(* CoDeSys 2.3 project: seven segment P1.pro *)
(* Libraries: STANDARD.LIB 25.11.03 12:18:06, IECSFC.LIB 25.11.03 12:18:06, ANALYZATION.LIB 25.11.03 12:18:06 *)

(* POU PLC_PRG, LD *)
PROGRAM PLC_PRG
VAR
	ix0: BOOL;
	a: WORD;
	count: CTUD;
END_VAR
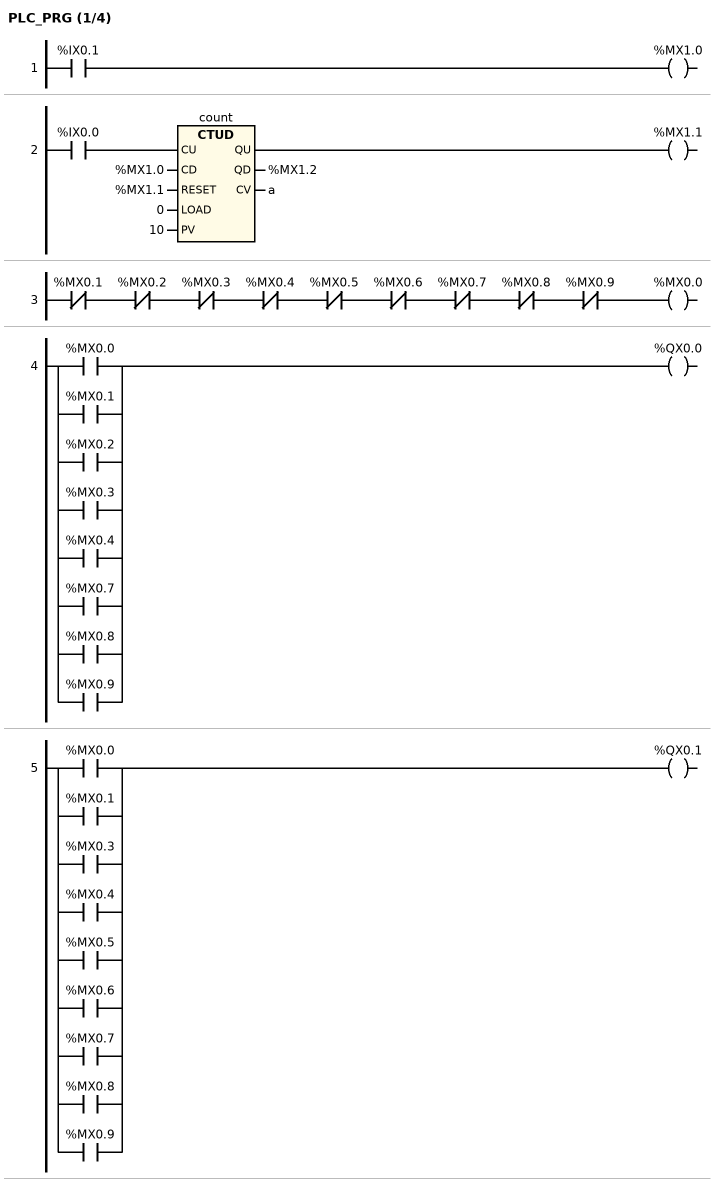
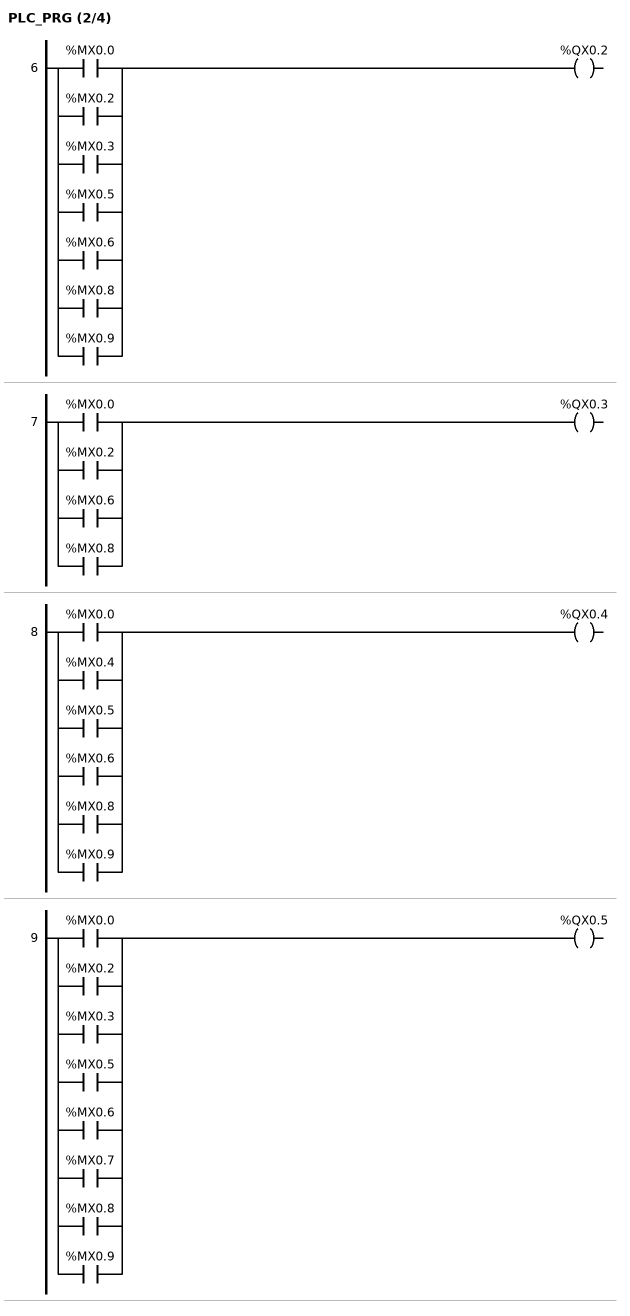
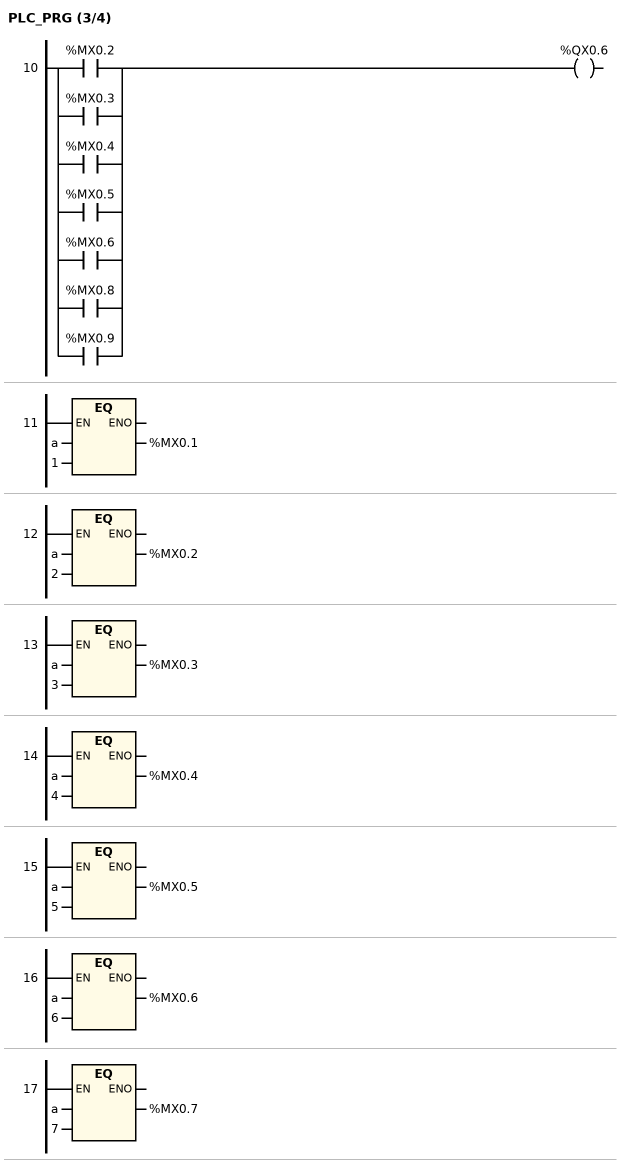
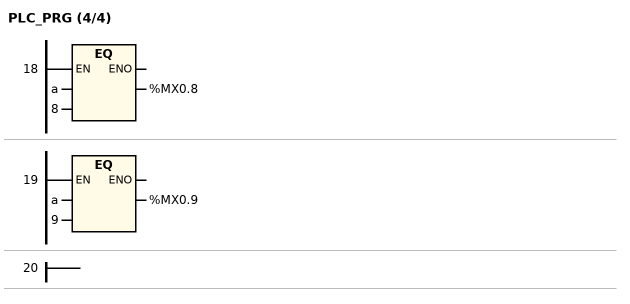
_LD_ (* Ladder Diagram *)
NETWORK 1
	[%IX0.1] --- (%MX1.0)
NETWORK 2
	[%IX0.0] - count:CTUD(CU: *, CD: %MX1.0, RESET: %MX1.1, LOAD: 0, PV: 10, QD => %MX1.2, CV => a) --- (%MX1.1)
NETWORK 3
	[/%MX0.1] - [/%MX0.2] - [/%MX0.3] - [/%MX0.4] - [/%MX0.5] - [/%MX0.6] - [/%MX0.7] - [/%MX0.8] - [/%MX0.9] --- (%MX0.0)
NETWORK 4
	{ [%MX0.0] | [%MX0.1] | [%MX0.2] | [%MX0.3] | [%MX0.4] | [%MX0.7] | [%MX0.8] | [%MX0.9] } --- (%QX0.0)
NETWORK 5
	{ [%MX0.0] | [%MX0.1] | [%MX0.3] | [%MX0.4] | [%MX0.5] | [%MX0.6] | [%MX0.7] | [%MX0.8] | [%MX0.9] } --- (%QX0.1)
NETWORK 6
	{ [%MX0.0] | [%MX0.2] | [%MX0.3] | [%MX0.5] | [%MX0.6] | [%MX0.8] | [%MX0.9] } --- (%QX0.2)
NETWORK 7
	{ [%MX0.0] | [%MX0.2] | [%MX0.6] | [%MX0.8] } --- (%QX0.3)
NETWORK 8
	{ [%MX0.0] | [%MX0.4] | [%MX0.5] | [%MX0.6] | [%MX0.8] | [%MX0.9] } --- (%QX0.4)
NETWORK 9
	{ [%MX0.0] | [%MX0.2] | [%MX0.3] | [%MX0.5] | [%MX0.6] | [%MX0.7] | [%MX0.8] | [%MX0.9] } --- (%QX0.5)
NETWORK 10
	{ [%MX0.2] | [%MX0.3] | [%MX0.4] | [%MX0.5] | [%MX0.6] | [%MX0.8] | [%MX0.9] } --- (%QX0.6)
NETWORK 11
	*
		EN --- EQ(a, 1) => %MX0.1
NETWORK 12
	*
		EN --- EQ(a, 2) => %MX0.2
NETWORK 13
	*
		EN --- EQ(a, 3) => %MX0.3
NETWORK 14
	*
		EN --- EQ(a, 4) => %MX0.4
NETWORK 15
	*
		EN --- EQ(a, 5) => %MX0.5
NETWORK 16
	*
		EN --- EQ(a, 6) => %MX0.6
NETWORK 17
	*
		EN --- EQ(a, 7) => %MX0.7
NETWORK 18
	*
		EN --- EQ(a, 8) => %MX0.8
NETWORK 19
	*
		EN --- EQ(a, 9) => %MX0.9
NETWORK 20
	*
_END_LD_
(* the same logic as Structured Text *)
(* Network 1 *)
%MX1.0 := %IX0.1;
(* Network 2 *)
count(CU := %IX0.0, CD := %MX1.0, RESET := %MX1.1, LOAD := 0, PV := 10);
%MX1.2 := count.QD;
a := count.CV;
%MX1.1 := count.QU;
(* Network 3 *)
%MX0.0 := NOT %MX0.1 AND NOT %MX0.2 AND NOT %MX0.3 AND NOT %MX0.4 AND NOT %MX0.5 AND NOT %MX0.6 AND NOT %MX0.7 AND NOT %MX0.8 AND NOT %MX0.9;
(* Network 4 *)
%QX0.0 := %MX0.0 OR %MX0.1 OR %MX0.2 OR %MX0.3 OR %MX0.4 OR %MX0.7 OR %MX0.8 OR %MX0.9;
(* Network 5 *)
%QX0.1 := %MX0.0 OR %MX0.1 OR %MX0.3 OR %MX0.4 OR %MX0.5 OR %MX0.6 OR %MX0.7 OR %MX0.8 OR %MX0.9;
(* Network 6 *)
%QX0.2 := %MX0.0 OR %MX0.2 OR %MX0.3 OR %MX0.5 OR %MX0.6 OR %MX0.8 OR %MX0.9;
(* Network 7 *)
%QX0.3 := %MX0.0 OR %MX0.2 OR %MX0.6 OR %MX0.8;
(* Network 8 *)
%QX0.4 := %MX0.0 OR %MX0.4 OR %MX0.5 OR %MX0.6 OR %MX0.8 OR %MX0.9;
(* Network 9 *)
%QX0.5 := %MX0.0 OR %MX0.2 OR %MX0.3 OR %MX0.5 OR %MX0.6 OR %MX0.7 OR %MX0.8 OR %MX0.9;
(* Network 10 *)
%QX0.6 := %MX0.2 OR %MX0.3 OR %MX0.4 OR %MX0.5 OR %MX0.6 OR %MX0.8 OR %MX0.9;
(* Network 11 *)
%MX0.1 := a = 1;
(* Network 12 *)
%MX0.2 := a = 2;
(* Network 13 *)
%MX0.3 := a = 3;
(* Network 14 *)
%MX0.4 := a = 4;
(* Network 15 *)
%MX0.5 := a = 5;
(* Network 16 *)
%MX0.6 := a = 6;
(* Network 17 *)
%MX0.7 := a = 7;
(* Network 18 *)
%MX0.8 := a = 8;
(* Network 19 *)
%MX0.9 := a = 9;
(* Network 20 *)
END_PROGRAM
